(* IEC 61131-3 sources: plc_generation_empirical_study/datasets/task_bank_c06_bounded_runtime_v0_2/tasks/C06_R08_lean_composite, 2 files *)

(* ---- interface.st ---- *)
FUNCTION_BLOCK C06_R08_lean_composite
VAR_INPUT
    A_Inspected : BOOL;
    A_Rejected : BOOL;
    A_Reset : BOOL;
    A_WindowSize : INT;
    A_RejectLimit : INT;
    B_S1 : BOOL;
    B_S2 : BOOL;
    B_S3 : BOOL;
    SubsystemBEnable : BOOL;
    CrossReset : BOOL;
END_VAR
VAR_OUTPUT
    A_WindowCount : INT;
    A_RejectCount : INT;
    A_LockedOut : BOOL;
    A_WindowComplete : BOOL;
    B_Vote : BOOL;
    B_Unanimous : BOOL;
    CrossReady : BOOL;
    CrossBlocked : BOOL;
END_VAR
END_FUNCTION_BLOCK

(* ---- reference.st ---- *)
FUNCTION_BLOCK C06_R08_lean_composite
VAR_INPUT
    A_Inspected : BOOL;
    A_Rejected : BOOL;
    A_Reset : BOOL;
    A_WindowSize : INT;
    A_RejectLimit : INT;
    B_S1 : BOOL;
    B_S2 : BOOL;
    B_S3 : BOOL;
    SubsystemBEnable : BOOL;
    CrossReset : BOOL;
END_VAR
VAR_OUTPUT
    A_WindowCount : INT;
    A_RejectCount : INT;
    A_LockedOut : BOOL;
    A_WindowComplete : BOOL;
    B_Vote : BOOL;
    B_Unanimous : BOOL;
    CrossReady : BOOL;
    CrossBlocked : BOOL;
END_VAR
VAR
    A_PrevInspected : BOOL := FALSE;
END_VAR

A_WindowComplete := FALSE;
IF A_Reset THEN
    A_WindowCount := 0;
    A_RejectCount := 0;
    A_LockedOut := FALSE;
ELSIF (NOT A_LockedOut) AND A_Inspected AND (NOT A_PrevInspected) THEN
    A_WindowCount := A_WindowCount + 1;
    IF A_Rejected THEN
        A_RejectCount := A_RejectCount + 1;
    END_IF;
    IF A_WindowCount >= A_WindowSize THEN
        IF A_RejectCount > A_RejectLimit THEN
            A_LockedOut := TRUE;
        END_IF;
        A_WindowCount := 0;
        A_RejectCount := 0;
        A_WindowComplete := TRUE;
    END_IF;
END_IF;
A_PrevInspected := A_Inspected;

IF CrossReset THEN
    CrossReady := FALSE;
ELSIF A_LockedOut THEN
    CrossReady := TRUE;
END_IF;
CrossBlocked := SubsystemBEnable AND (NOT CrossReady);

IF SubsystemBEnable AND CrossReady THEN
    B_Vote := (B_S1 AND B_S2) OR (B_S1 AND B_S3) OR (B_S2 AND B_S3);
    B_Unanimous := (B_S1 AND B_S2 AND B_S3) OR ((NOT B_S1) AND (NOT B_S2) AND (NOT B_S3));
ELSE
    B_Vote := FALSE;
    B_Unanimous := FALSE;
END_IF;

END_FUNCTION_BLOCK
